// Mitsubishi GX Works2 project: MPS 장비 제어하기 2_2   PLC: Q03UDV

PROGRAM MAIN
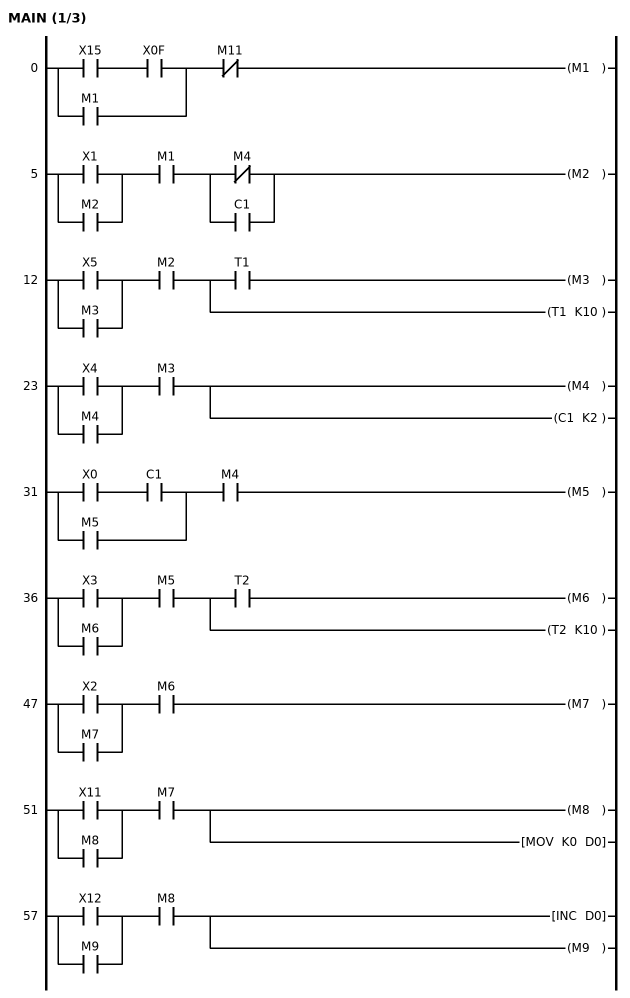
0     LD      X15
      AND     X0F
      OR      M1
      ANI     M11
      OUT     M1
5     LD      X1
      OR      M2
      AND     M1
      LDI     M4
      OR      C1
      ANB
      OUT     M2
12    LD      X5
      OR      M3
      AND     M2
      MPS
      AND     T1
      OUT     M3
      MPP
      OUT     T1 K10
23    LD      X4
      OR      M4
      AND     M3
      OUT     M4
      OUT     C1 K2
31    LD      X0
      AND     C1
      OR      M5
      AND     M4
      OUT     M5
36    LD      X3
      OR      M6
      AND     M5
      MPS
      AND     T2
      OUT     M6
      MPP
      OUT     T2 K10
47    LD      X2
      OR      M7
      AND     M6
      OUT     M7
51    LD      X11
      OR      M8
      AND     M7
      OUT     M8
      MOV     K0 D0
57    LD      X12
      OR      M9
      AND     M8
      INC     D0
      OUT     M9
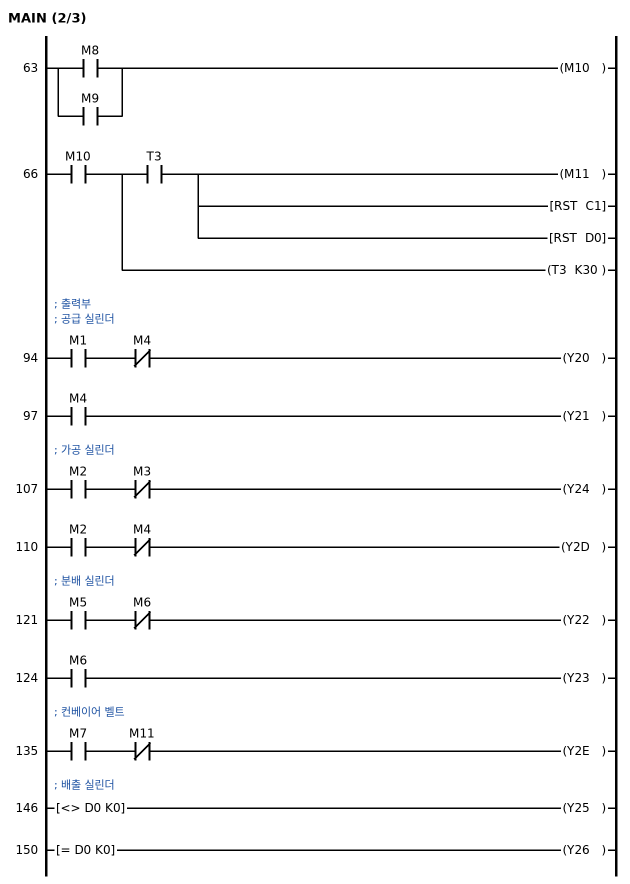
63    LD      M8
      OR      M9
      OUT     M10
66    LD      M10
      MPS
      AND     T3
      OUT     M11
      RST     C1
      RST     D0
      MPP
      OUT     T3 K30
; 출력부
; 공급 실린더
94    LD      M1
      ANI     M4
      OUT     Y20
97    LD      M4
      OUT     Y21
; 가공 실린더
107   LD      M2
      ANI     M3
      OUT     Y24
110   LD      M2
      ANI     M4
      OUT     Y2D
; 분배 실린더
121   LD      M5
      ANI     M6
      OUT     Y22
124   LD      M6
      OUT     Y23
; 컨베이어 벨트
135   LD      M7
      ANI     M11
      OUT     Y2E
; 배출 실린더
146   LD<>    D0 K0
      OUT     Y25
150   LD=     D0 K0
      OUT     Y26
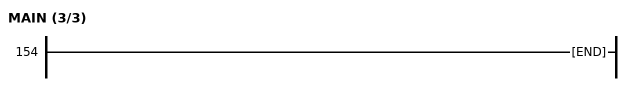
154   END
END_PROGRAM
